Staubli VAL3: restartMove.pgx

public program restartMove()
begin
  restartMove()
end
